// TIA Portal V17 export
// export: Created 2021-12-03T08:13:08.2140584Z, ExportSetting WithDefaults, DisplayName Totally Integrated Automation Portal, DisplayVersion V17, DisplayName TIA Portal Openness, DisplayVersion V17, DisplayName TIA Portal Version Control Interface, DisplayVersion V17, DisplayName STEP 7 Professional, DisplayVersion V17, DisplayName STEP 7 Safety, DisplayVersion V17, DisplayName WinCC Advanced, DisplayVersion V17
FUNCTION_BLOCK "FB_FitMem"   // FB40, FBD
VERSION : 0.1
// stored: AutoNumber false, IsIECCheckEnabled false, UDAEnableTagReadback false
   VAR_INPUT
      I_Ack : Bool;
      I_Fit : Bool;
   END_VAR
   VAR_OUTPUT
      O_Fit : Bool;
      O_AskRq : Bool;
   END_VAR
   VAR DB_SPECIFIC
      S_AxVar_Pedg_Ack : Bool;
      S_AxVar_RSFF_Flt : Bool;
      S_Flt : Bool;
   END_VAR
   VAR_TEMP   // added for the SCL form of the ladder/FBD networks
      _w1 : Bool;
   END_VAR
BEGIN

REGION Network 1
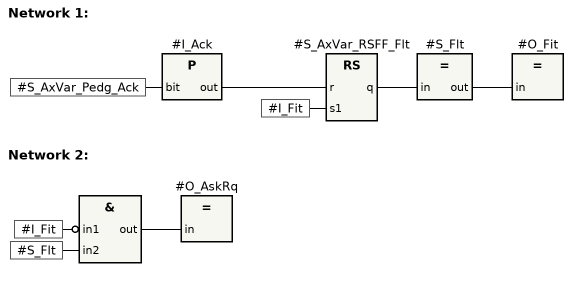
   #_w1 := #I_Ack AND NOT #S_AxVar_Pedg_Ack;   // rising edge of #I_Ack
   #S_AxVar_Pedg_Ack := #I_Ack;
   IF #_w1 THEN
       #S_AxVar_RSFF_Flt := FALSE;   // RS flip-flop
   END_IF;
   IF #I_Fit THEN #S_AxVar_RSFF_Flt := TRUE; END_IF;
   #S_Flt := #S_AxVar_RSFF_Flt;
   #O_Fit := #S_AxVar_RSFF_Flt;
END_REGION

REGION Network 2
   #O_AskRq := NOT #I_Fit AND #S_Flt;
END_REGION
END_FUNCTION_BLOCK
